// TIA Portal project "example_project" (V17)

(* hardware
DEVICE "S7-1500/ET200MP station_1"  S7-1500 station
   slot 0: "Rail_0"  Rack  6ES7 590-1***0-0AA0
   slot 1: "PLC_1"  CPU 1515F-2 PN  6ES7 515-2FM01-0AB0  V2.8
      slot 3: "CPU display_1"  6ES7591-1BA00-0AA0
      slot 32768: "PROFINET interface_1"  X1
         slot 32769: "Port_1"  X1 P1
         slot 32770: "Port_2"  X1 P2
      slot 33024: "PROFINET interface_2"  X2
         slot 33025: "Port_1"  X2 P1
      slot 34817: "Virtual CP interface port_1"  Virtual CP interface port  Virtual CP interface port
*)

// ===== PLC "PLC_1"  CPU 1515F-2 PN =====

VAR_GLOBAL   // PLC tag table "Default tag table"
   "TakeReferenceSnapshot" AT %I0.0 : Bool;
END_VAR

DATA_BLOCK "Main_Safety_RTG1_DB"   // DB1, F_DB
{ S7_Optimized_Access := 'TRUE' }
NAME : FUSI
VERSION : 0.1
// stored: InstanceOfName Main_Safety_RTG1
"Main_Safety_RTG1"
BEGIN
END_DATA_BLOCK

DATA_BLOCK "SickCamera_DB"   // DB2
{ S7_Optimized_Access := 'FALSE' }
VERSION : 0.1
// stored: InstanceOfName SickCamera
"SickCamera"
BEGIN
END_DATA_BLOCK

FUNCTION_BLOCK "Main_Safety_RTG1"   // FB1, F_FBD
{ S7_Optimized_Access := 'TRUE' }
BEGIN
END_FUNCTION_BLOCK

FUNCTION_BLOCK "SickCamera"   // FB2, LAD
{ S7_Optimized_Access := 'FALSE' }
VERSION : 0.1
   VAR
      CurrentImage : Array[0..#ImageSize] of UDInt;
      CurrentAverage : UDInt;
      DifferenceOut : Real;
   END_VAR
   VAR_TEMP
      ReferenceImage : Array[0..#ImageSize] of UDInt;
      DifferencePercentage : Real;
   END_VAR
   VAR CONSTANT
      Low : UDInt := 15;   // mm
      High : UDInt := 4000;   // mm
      ImageSize : UDInt := 1296;
   END_VAR
BEGIN

REGION Network 1
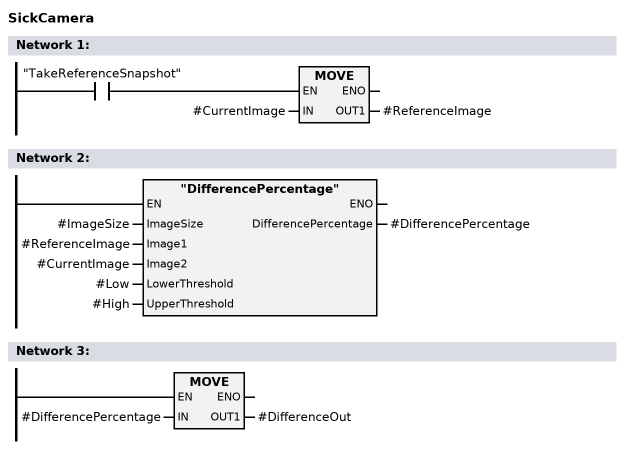
   RUNG wire#powerrail
      Contact( "TakeReferenceSnapshot" )
      Move(in := #CurrentImage, out1 => #ReferenceImage)
   END_RUNG
   // the same network as SCL:
   IF "TakeReferenceSnapshot" THEN #ReferenceImage := #CurrentImage; END_IF;
END_REGION

REGION Network 2
   RUNG wire#powerrail
      "DifferencePercentage"(ImageSize := #ImageSize, Image1 := #ReferenceImage, Image2 := #CurrentImage, LowerThreshold := #Low, UpperThreshold := #High, DifferencePercentage => #DifferencePercentage)
   END_RUNG
   // the same network as SCL:
   "DifferencePercentage"(ImageSize := #ImageSize,
                          Image1 := #ReferenceImage,
                          Image2 := #CurrentImage,
                          LowerThreshold := #Low,
                          UpperThreshold := #High,
                          DifferencePercentage => #DifferencePercentage);
END_REGION

REGION Network 3
   RUNG wire#powerrail
      Move(in := #DifferencePercentage, out1 => #DifferenceOut)
   END_RUNG
   // the same network as SCL:
   #DifferenceOut := #DifferencePercentage;
END_REGION
END_FUNCTION_BLOCK

FUNCTION "DifferencePercentage" : Void   // FC1, SCL
{ S7_Optimized_Access := 'TRUE' }
VERSION : 0.1
   VAR_INPUT
      ImageSize : UDInt;
      Image1 : Array[*] of UDInt;
      Image2 : Array[*] of UDInt;
      LowerThreshold : UDInt;
      UpperThreshold : UDInt;
   END_VAR
   VAR_OUTPUT
      DifferencePercentage : Real;
   END_VAR
   VAR_TEMP
      Index : UDInt;
      Delta : DInt;
      DifferenceCount : UDInt;
   END_VAR
BEGIN
   #DifferenceCount := 0;
   IF #ImageSize > 0 THEN
       FOR #Index := 1 TO #ImageSize DO
           #Delta := ABS_DINT(#Image1[#Index] - #Image2[#Index]);
           IF #Delta >= #LowerThreshold AND #Delta <= #UpperThreshold THEN
               #DifferenceCount := #DifferenceCount + 1;
           END_IF;
       END_FOR;

       #DifferencePercentage := (UDINT_TO_REAL(#DifferenceCount) / UDINT_TO_REAL(#ImageSize)) * 100.0;
   END_IF;
END_FUNCTION

ORGANIZATION_BLOCK "Main"   // OB1, LAD, ProgramCycle
TITLE = "Main Program Sweep (Cycle)"
{ S7_Optimized_Access := 'TRUE' }
VERSION : 0.1
   VAR_INPUT
      Initial_Call : Bool;   // Initial call of this OB
      Remanence : Bool;   // =True, if remanent data are available
   END_VAR
BEGIN

REGION Network 1
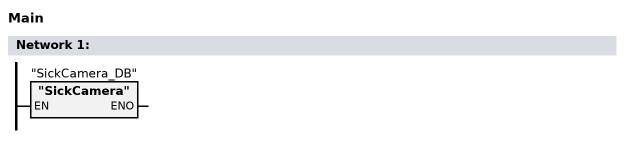
   RUNG wire#powerrail
      "SickCamera_DB"()
   END_RUNG
   // the same network as SCL:
   "SickCamera_DB"();   // "SickCamera"
END_REGION
END_ORGANIZATION_BLOCK